(* IEC 61131-3 sources: repolevel_ST_code_completion/dataset/project_code/measurement_control/PRG, 1 file *)

(* ---- PLC_PRG.st ---- *)
PROGRAM PLC_PRG
VAR
	Tank01 : Tank;
END_VAR

Tank01(stName:='Tank01',nMaxLevel:=99, nMinLevel:=0,nMaxTemp:=55, nMinTemp:=44);
